FUNCTION_BLOCK FB_LightBase IMPLEMENTS I_LightBase

VAR
	sName				: STRING;
	sAddress			: STRING;
	bState				: BOOL;
	nLightID			: USINT;
END_VAR

PROPERTY ID : USINT
GET
ID := nLightID;
END_GET
SET
nLightID := ID;
END_SET
END_PROPERTY

PROPERTY PUBLIC State : BOOL
GET
State := bState;
END_GET
SET
bState := State;
END_SET
END_PROPERTY

METHOD Toggle
IF NOT bState THEN
	THIS^.TurnON();
ELSE
	THIS^.TurnOFF();
END_IF
END_METHOD

METHOD TurnOFF
THIS^.bState := FALSE;
END_METHOD

METHOD TurnON
THIS^.bState := TRUE;
END_METHOD

END_FUNCTION_BLOCK

(* stored: Version 1.1.0.1, ProductVersion 3.1.4024.12
   POU FB_LightBase: Id {ee94f5f8-49a0-4004-80b5-30dbbdf9bbd0}, SpecialFunc None
   Property ID: Id {97549fe9-26e8-47be-9c3e-102e6b2b0fcd}
   Get Get: Id {75de85c8-a22f-4e91-a3b0-ab4c41e69f8e}
   Set Set: Id {f68e7ef6-0a59-43b8-8082-d5d4536719aa}
   Property State: Id {25721263-ebdb-4ddb-bee8-5daa2e6c7902}
   Get Get: Id {e0f5c6fd-9025-45f7-ad22-1a48dcc53242}
   Set Set: Id {727318e8-ea11-4911-bef6-80c4799add69}
   Method Toggle: Id {f94300be-42bc-492e-b93c-ad7b802327d9}
   Method TurnOFF: Id {4ffa847b-646b-4ec6-83a7-8fe43eb89af7}
   Method TurnON: Id {2f5892f3-5587-43be-bc99-96832e112373} *)
